FUNCTION_BLOCK IO_RouteAO (* Backend router for IO_AO: 0 simulated, 1 local IO handle, 2 Modbus *)
  (* Standard: 61499-2 *)
  (* Version 0.1, 2026-09-28, Project contributors, AAU Smart Production Lab *)
  PACKAGE modlib;
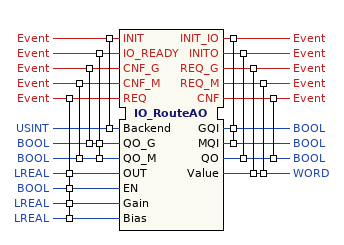
  EVENT_INPUT
    INIT WITH Backend;
    IO_READY WITH QO_G, QO_M;
    CNF_G WITH QO_G;
    CNF_M WITH QO_M;
    REQ WITH OUT, EN, Gain, Bias;
  END_EVENT
  EVENT_OUTPUT
    INIT_IO WITH GQI, MQI;
    INITO WITH QO;
    REQ_G WITH Value;
    REQ_M WITH Value;
    CNF WITH QO;
  END_EVENT
  VAR_INPUT
    Backend : USINT;
    QO_G : BOOL;
    QO_M : BOOL;
    OUT : LREAL;
    EN : BOOL;
    Gain : LREAL := 1.0;
    Bias : LREAL;
  END_VAR
  VAR_OUTPUT
    GQI : BOOL;
    MQI : BOOL;
    QO : BOOL;
    Value : WORD;
  END_VAR
  VAR
    Raw : LREAL;
  END_VAR
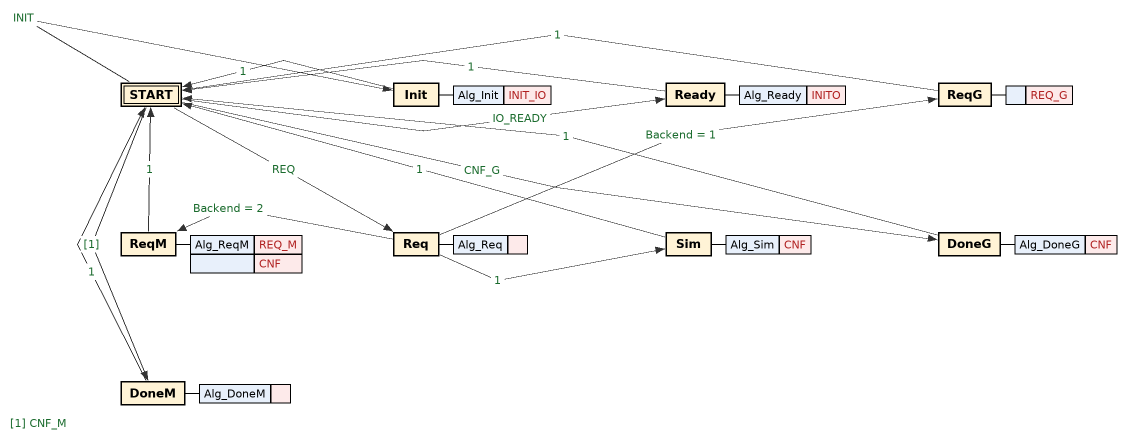
  EC_STATES
    START;
    Init : Alg_Init -> INIT_IO;
    Ready : Alg_Ready -> INITO;
    ReqG : -> REQ_G;
    ReqM : Alg_ReqM -> REQ_M, -> CNF;
    Req : Alg_Req;
    Sim : Alg_Sim -> CNF;
    DoneG : Alg_DoneG -> CNF;
    DoneM : Alg_DoneM;
  END_STATES
  EC_TRANSITIONS
    START TO Init := INIT;
    Init TO START := 1;
    START TO Ready := IO_READY;
    Ready TO START := 1;
    START TO Req := REQ;
    Req TO ReqG := Backend = 1;
    Req TO ReqM := Backend = 2;
    Req TO Sim := 1;
    START TO DoneG := CNF_G;
    START TO DoneM := CNF_M;
    ReqG TO START := 1;
    ReqM TO START := 1;
    Sim TO START := 1;
    DoneG TO START := 1;
    DoneM TO START := 1;
  END_TRANSITIONS
  ALGORITHM Alg_Init IN ST:
GQI := Backend = 1;
MQI := Backend = 2;
  END_ALGORITHM
  ALGORITHM Alg_Ready IN ST:
QO := (Backend = 0) OR ((Backend = 1) AND QO_G) OR ((Backend = 2) AND QO_M);
  END_ALGORITHM
  ALGORITHM Alg_ReqM IN ST:
QO := QO_M;
  END_ALGORITHM
  ALGORITHM Alg_Req IN ST:
IF EN THEN
  Raw := Bias + OUT * Gain;
  IF Raw < 0.0 THEN
    Raw := 0.0;
  ELSIF Raw > 65535.0 THEN
    Raw := 65535.0;
  END_IF;
  Value := UINT_TO_WORD(LREAL_TO_UINT(Raw));
ELSE
  Value := WORD#0;
END_IF;
  END_ALGORITHM
  ALGORITHM Alg_Sim IN ST:
QO := TRUE;
  END_ALGORITHM
  ALGORITHM Alg_DoneG IN ST:
QO := QO_G;
  END_ALGORITHM
  ALGORITHM Alg_DoneM IN ST:
QO := QO_M;
  END_ALGORITHM
END_FUNCTION_BLOCK
